(* Logix 5000 project; controller Prueba2 vendor 1 type 14 code 156 rev 30.11; software revision 30.00 *)

TASK MainTask (continuous, watchdog 500 ms) : MainProgram

MODULES
   Local : vendor 1 type 14 code 156 (Compact 0, rev 30.11)
      DI_4 : 1769-IQ16 (Compact 4, rev 1.1, Input RPI 20 ms)
      DO_5 : vendor 1 type 7 code 86 (Compact 5, rev 2.1, Output RPI 20 ms)
END_MODULES

PROGRAM MainProgram   (* main routine MainRoutine *)
VAR
   MOTOR : ALIAS FOR Local:5:O.Data.0;
   start : ALIAS FOR Local:4:I.Data.1;
   stop : ALIAS FOR Local:4:I.Data.0;
END_VAR

ROUTINE MainRoutine   (* ladder *)
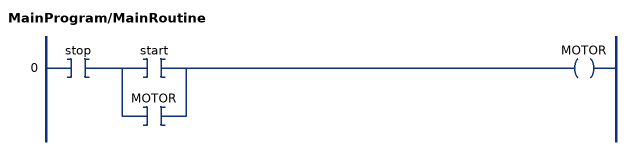
   0: XIC(stop)[XIC(start) ,XIC(MOTOR) ]OTE(MOTOR);
END_ROUTINE
END_PROGRAM
